FUNCTION TryConvert_DINT_TO_DWORD : BOOL
VAR_INPUT
	in : DINT;
	out : REFERENCE TO DWORD;
END_VAR

IF in < DatatypeLimits.MIN_VALUE_OF_DINT_WHICH_CAN_BE_HELD_IN_A_DWORD THEN
	RETURN;
END_IF

out := DINT_TO_DWORD(in);
TryConvert_DINT_TO_DWORD := TRUE;

END_FUNCTION

(* stored: Version 1.1.0.1, ProductVersion 3.1.4024.12
   POU TryConvert_DINT_TO_DWORD: Id {074b9e40-25f6-4168-b6ed-92da3522c211}, SpecialFunc None *)
